// Mitsubishi GX Works2 project: SEQUENCE_REPEAT1   PLC: Q03UDV

PROGRAM MAIN
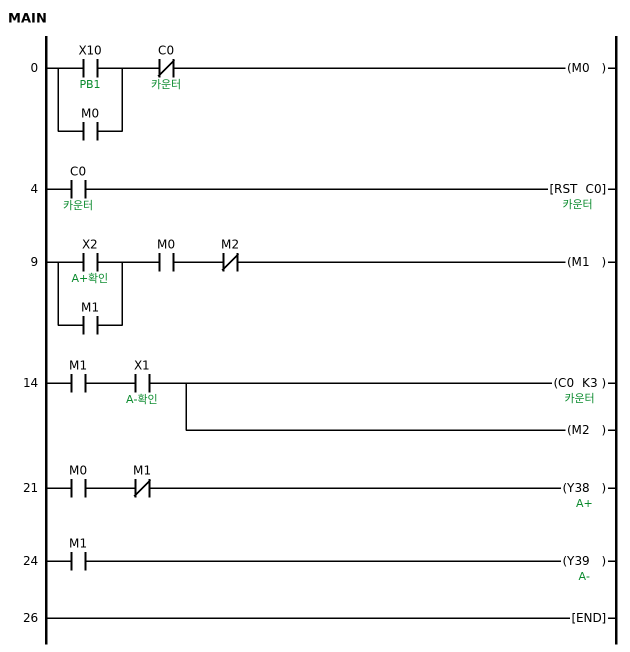
0     LD      X10  ; PB1
      OR      M0
      ANI     C0  ; 카운터
      OUT     M0
4     LD      C0  ; 카운터
      RST     C0  ; 카운터
9     LD      X2  ; A+확인
      OR      M1
      AND     M0
      ANI     M2
      OUT     M1
14    LD      M1
      AND     X1  ; A-확인
      OUT     C0 K3  ; 카운터
      OUT     M2
21    LD      M0
      ANI     M1
      OUT     Y38  ; A+
24    LD      M1
      OUT     Y39  ; A-
26    END
END_PROGRAM
